{attribute addProperty BoxType "KL3021"}
{attribute addProperty Id "Channel_1Channel_B0A8062F00"}
{attribute addProperty CRC "2809087995"}
{attribute addProperty SizeInBites "0"}
{attribute addProperty SizeInBytes "0"}
TYPE KL3021_A76F47FB :
STRUCT
	{attribute addProperty Name "Channel_1"}
	Channel_1 : Channel_B0A8062F;
END_STRUCT
END_TYPE

(* stored: Version 1.2.0.0, ProductVersion 3.1.4024.9
   DUT KL3021_A76F47FB: Id {f3c19940-fcd5-41dd-9a7c-2767ae82326f} *)
